FUNCTION_BLOCK TestMachine
VAR
	idleState : State(name := 'Idle');
	runningState : State(name := 'Running');
	stoppedState : State(name := 'Stopped');
	abortedState : State(name := 'Aborted');
	
	t2 : Transition(event := TestMachineEvents.Start, sourceState := idleState, destinationState := runningState);
	t1 : Transition(event := TestMachineEvents.Stop, sourceState := runningState, destinationState := stoppedState);
	t3 : Transition(event := TestMachineEvents.Abort, sourceState := idleState, destinationState := abortedState);
	t4 : Transition(event := TestMachineEvents.Abort, sourceState := runningState, destinationState := abortedState);
	t5 : Transition(event := TestMachineEvents.Abort, sourceState := stoppedState, destinationState := abortedState);
	t6 : Transition(event := TestMachineEvents.Reset, sourceState := stoppedState, destinationState := idleState);
	t7 : Transition(event := TestMachineEvents.Clear, sourceState := abortedState, destinationState := IdleState);
	
	tl1 : TransitionList(t1, 0);
	tl2 : TransitionList(t2, tl1);
	tl3 : TransitionList(t3, tl2);
	tl4 : TransitionList(t4, tl3);
	tl5 : TransitionList(t5, tl4);
	tl6 : TransitionList(t6, tl5);
	tl7 : TransitionList(t7, tl6);
	
	fsm : FSM(defaultState := idleState, transitions := tl7);
END_VAR

METHOD Abort
VAR_INPUT
END_VAR
fsm.Event(TestMachineEvents.Abort);
END_METHOD

METHOD Clear
fsm.Event(TestMachineEvents.Clear);
END_METHOD

PROPERTY CurrentStateName : STRING
GET
CurrentStateName := fsm.CurrentState.Name;
END_GET
END_PROPERTY

METHOD Reset
fsm.Event(TestMachineEvents.Reset);
END_METHOD

METHOD Start
fsm.Event(TestMachineEvents.Start);
END_METHOD

METHOD Stop
fsm.Event(TestMachineEvents.Stop);
END_METHOD

END_FUNCTION_BLOCK

(* stored: Version 1.1.0.1, ProductVersion 3.1.4024.12
   POU TestMachine: Id {8b5ec37e-8862-0370-1ebd-55ab2aab7536}, SpecialFunc None
   Method Abort: Id {953cbf8d-b997-0fa3-1be9-e595a0db8ff1}
   Method Clear: Id {6b7c39d1-a0a2-04ea-0fa2-3ea744929cfb}
   Property CurrentStateName: Id {caa27d60-67f5-06b8-145e-377dbcc4d634}
   Get Get: Id {0ce5915d-a6ed-071e-38ae-d6ed542ce3be}
   Method Reset: Id {d5e64aa2-5467-0e48-2a4f-6f2b51e34206}
   Method Start: Id {9d261092-ac5f-02c2-0728-62d6a9a253f0}
   Method Stop: Id {ae065239-f384-02d3-327d-8b491fa1362b} *)
